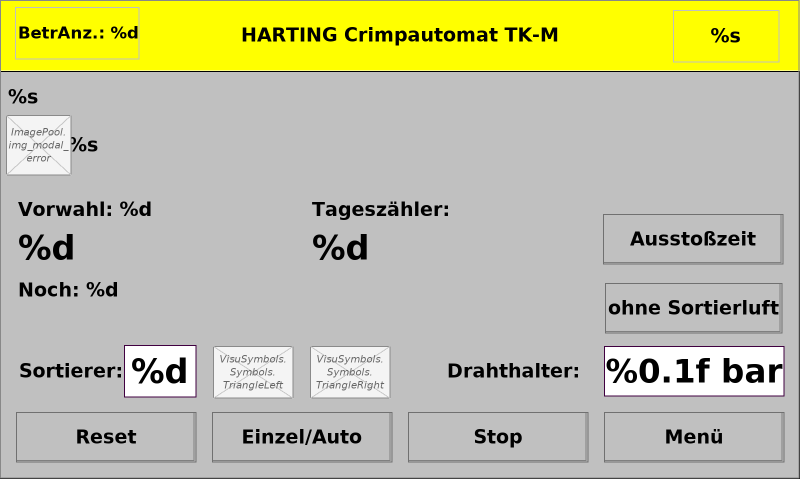
VISUALIZATION Start  // 800x479
    Rectangle (0,71 800x408)
    Rectangle (0,0 800x70), "HARTING Crimpautomat TK-M"
    Rectangle (15,192 284x35), "Vorwahl: %d", text variable: DB6.diStueck_Vorwahl
    Rectangle (15,270 191x40), "Noch: %d", text variable: DB6.diStueck_Noch
    Rectangle (15,225 291x45), "%d", text variable: DB6.diStueck_Fertig
    Rectangle (309,192 284x35), "Tageszähler:"
    Rectangle (309,225 262x45), "%d", text variable: DB6.diStueck_Fertig
    Button (16,412 180x50), "Reset"
        OnMouseClick: execute { P_OnResetClick(); }
    Button (212,412 180x50), "Einzel/Auto", colour toggle: VAT.bEinzelSchritt
        OnMouseClick: execute { F_AuswertungBefehlstastenVonTP(tastenWert := 30); }
    Button (408,412 180x50), "Stop"
        OnMouseClick: execute { F_AuswertungBefehlstastenVonTP(tastenWert := CVL.BTN_STOP); }
    Button (604,412 180x50), "Menü"
        OnMouseUp: change screen: Menu
    Rectangle (124,345 72x52), "%d", text variable: DB6.iSortierer
        OnMouseClick: write the text variable via VisuDialogs.Numpad, min 0, max 100, title 'Sortierer'
    Rectangle (16,346 106x50), "Sortierer:"
    Image (213,346 80x52), image: VisuSymbols.Symbols.TriangleLeft
        OnMouseClick: execute { P_DecSollRuettel(); }
    Image (310,346 80x52), image: VisuSymbols.Symbols.TriangleRight
        OnMouseClick: execute { P_IncSollRuettel(); }
    Button (603,214 180x50), "Ausstoßzeit", invisible if: DB6.rAusstossverz > -0.05 AND DB6.rAusstossverz < 0.05
        OnMouseUp: change screen: Ausstossverz
    Rectangle (441,346 145x50), "Drahthalter:"
    Button (605,283 177x50), "ohne Sortierluft", text list: 'BetrAnzeigeListe', text index: VAT.sortierTextID
        OnMouseUp: execute { VAT.bSortiererBlasen := NOT VAT.bSortiererBlasen; }
    Rectangle (604,346 180x50), "%0.1f bar", text variable: DB6.rDrahthalterSchliessdruck
    Rectangle (673,10 106x52), "%s", text variable: VisuElems.CurrentLanguage, invisible if: TRUE
    Rectangle (5,77 791x40), "%s", invisible if: GVL.zeigeFehler, text list: 'BetrAnzeigeListe', text index: DB6.w226_Betr_Anz_Wert
    Rectangle (15,7 124x52), "BetrAnz.: %d", text variable: DB6.w226_Betr_Anz_Wert, invisible if: TRUE
    Rectangle (65,125 730x40), "%s", invisible if: NOT GVL.zeigeFehler, text list: 'BetrAnzeigeListe', text index: GVL.SolPosErrorIdx
    Image (6,115 65x60), invisible if: NOT GVL.zeigeFehler, image: ImagePool.img_modal_error
        OnMouseUp: execute { RVL.e12Online := NOT RVL.e12Online; }
END_VISUALIZATION

(* stored: Version 1.1.0.1, ProductVersion 3.1.4024.3
   Visu Start: Id {81cf644b-f21d-4337-a6b5-886c3fc38555} *)
